Universal Robots PolyScope program: leftright.urp

Program leftright (createdIn=3.4.4.412 lastSavedIn=3.4.4.412 directory=/programs installation=default robotSerialNumber=2017356443)
Calibrated DH parameters: a=[0.000092, -0.116521, -0.182101, -0.000106, 0.000044, 0]; d=[0.089391, 255.189113, -82.629387, -172.449369, 0.094782, 0.082637]; alpha=[1.569598, 0.001603, 0.002015, 1.570234, -1.570307, 0]; deltaTheta=[-0.000017, 1.293309, -0.204843, -1.088417, 0.000036, -0.000078]
Robot Program (runOnlyOnce=false motionType=MoveJ speed=1.047198 acceleration=1.396263 useActiveTCP=false)
  MoveJ speed 60 deg/s, acceleration 80 deg/s^2 (useActiveTCP=false)
    Waypoint Waypoint_1: TCP in base x=439.538 y=-427.735 z=432.169 mm, rx=1.1592 ry=-1.0861 rz=0.4722 rad; joints [-25.793, -107.843, -70.494, -142.73, -0.101, 21.468] deg
  Wait Sleep waitTime=1
  MoveJ speed 60 deg/s, acceleration 80 deg/s^2 (useActiveTCP=false)
    Waypoint Waypoint_2: TCP in base x=611.193 y=51.104 z=432.175 mm, rx=1.5994 ry=-0.5394 rz=1.1263 rad; joints [23.206, -107.843, -70.494, -142.73, -0.101, 21.468] deg
  Wait Sleep waitTime=1
